FUNCTION_BLOCK Q_ChangePolygonScale (* Command Change Polygon Scale( Part 6 - F.54 ) *)
  (* Standard: ISO 11783-6; Description: see Description Tab *)
  (* Version 1.0, 2022-07-08, franz *)
  (* Documentation:
  Command Change Polygon Scale( Part 6 - F.54 )
   This command is used by a Working Set to change the scale of a complete Output Polygon object.
   param[in] {objectID, uint16_t}
   Object ID of the Output Polygon object to scale
   param[in] {widthAttribute, uint16_t}
   New width attribute
   param[in] {heightAttribute, uint16_t}
   New height attribute
   Return Values: 
   int16_t
    - VT_E_NO_ERR (0) - OK
   - VT_E_OVERFLOW (-6) - buffer overflow
   - VT_E_NOACT (-8) - Command not possible in current state
   - VT_E_NO_INSTANCE (-21) - No VT client available
   - VT_E_ISO_INSTANCE_INVALID (-129) - Identifier for instance (connection) invalid
   - VT_E_NOT_ALVIE (-130) - Identifier for instance valid, but VT Dead.
  *)
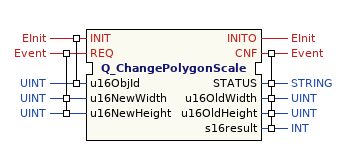
  EVENT_INPUT
    INIT : EInit WITH u16ObjId; (* Service Initialization *)
    REQ WITH u16NewWidth, u16NewHeight; (* Service Request *)
  END_EVENT
  EVENT_OUTPUT
    INITO : EInit; (* Initialization Confirm *)
    CNF WITH STATUS, s16result, u16OldWidth, u16OldHeight; (* Confirmation of Requested Service *)
  END_EVENT
  VAR_INPUT
    u16ObjId : UINT; (* Object ID of the Output Polygon object to change *)
    u16NewWidth : UINT; (* New width attribute *)
    u16NewHeight : UINT; (* New height attribute *)
  END_VAR
  VAR_OUTPUT
    STATUS : STRING; (* Service Status *)
    u16OldWidth : UINT; (* Old width attribute *)
    u16OldHeight : UINT; (* Old height attribute *)
    s16result : INT; (* retval see description *)
  END_VAR
END_FUNCTION_BLOCK
